# EPICS autosave request: ADRIXSCam/iocs/rixscamIOC/iocBoot/iocRixsCam/auto_settings.req
file "rixscam_settings.req",    P=$(P),  R=cam1:
file "NDStdArrays_settings.req",    P=$(P), R=image1:
file "commonPlugin_settings.req",   P=$(P)
